// TwinCAT 3 PLC project PersistentData
// Title: ManagePersistentData
// Company: beckhoff.co.jp
// Author: Beckhoff Automation K.K.
// ProjectVersion: 1.0.0.1
// ProgramVersion: 3.1.4024.0
// libraries:
//   Tc2_IoFunctions, * (Beckhoff Automation GmbH)
//   Tc2_Standard, * (Beckhoff Automation GmbH)
//   Tc2_SUPS, * (Beckhoff Automation GmbH)
//   Tc2_System, * (Beckhoff Automation GmbH)
//   Tc2_Utilities, * (Beckhoff Automation GmbH)
//   Tc3_Module, * (Beckhoff Automation GmbH)
// project tree:
//   DUTs/ E_ShutdownMode.TcDUT, E_UPSState.TcDUT
//   / PlcTask.TcTTO
//   POUs/ FB_GenericUPS.TcPOU, FB_ShutDown.TcPOU, FB_SUPS_CX51x0.TcPOU, FB_UPS_STUB.TcPOU, iUPS.TcIO, MAIN.TcPOU
//   Project Information/ F_GetCompany.TcPOU, F_GetTitle.TcPOU, F_GetVersion.TcPOU
//   Version/ Global_Version.TcGVL
// real-time tasks:
//   TASK PlcTask: cycle T#10ms, priority 20, ADS port 350

CONFIGURATION PersistentData
    RESOURCE PLC ON TwinCAT3
        TASK PlcTask(INTERVAL := T#10ms, PRIORITY := 20);
        PROGRAM MAIN WITH PlcTask : MAIN;
    END_RESOURCE
END_CONFIGURATION

// ---- DUTs/E_ShutdownMode.TcDUT
{attribute 'qualified_only'}
{attribute 'strict'}
TYPE E_ShutdownMode :
(
	init := 0,			// system is working
	persistent_data,	// persist data
	shutting_down		// system shutting down
);
END_TYPE

// ---- DUTs/E_UPSState.TcDUT
{attribute 'qualified_only'}
{attribute 'strict'}
TYPE E_UPSState :
(
	init := 0,		// UPS not working
	on_power,		// power supplied normally
	on_battery,		// continue working on battery
	critical_error,	// system shutdown
	facility_error	// UPC failure
);
END_TYPE

// ---- Version/Global_Version.TcGVL
{attribute 'TcGenerated'}
{attribute 'no-analysis'}
{attribute 'linkalways'}
// This function has been automatically generated from the project information.
VAR_GLOBAL CONSTANT
	{attribute 'const_non_replaced'}
	stLibVersion_ManagePersistentData : ST_LibVersion := (iMajor := 1, iMinor := 0, iBuild := 0, iRevision := 1, nFlags := 0, sVersion := '1.0.0.1');
END_VAR

// ---- POUs/iUPS.TcIO
INTERFACE iUPS

(*
Method of saving persistent data
=================================================

Author
	: Takashi Ichihashi

Date
	: 02 Aug, 2023

Overview
===============

This method is assumed that persistent values are saved when ups running without online power.
"WritePersistentData" FB has to be executed explicily in case of GenericUPS is used. You might define this FB instance on this method.
If you use "SUPS", it might be saved persistent data automatically when power failed, so nothing need to be defined on this method.

*)
METHOD persist_data : BOOL
VAR_INPUT
END_VAR
END_METHOD

METHOD shutdown : BOOL
VAR_INPUT
END_VAR
END_METHOD

PROPERTY shutdown_delay : TIME
GET
END_GET
SET
END_SET
END_PROPERTY

PROPERTY UPSState : E_UPSState
GET
END_GET
END_PROPERTY

METHOD watch_status : BOOL
VAR_INPUT
END_VAR
END_METHOD

END_INTERFACE

// ---- POUs/MAIN.TcPOU
PROGRAM MAIN
VAR
	fbShutdown	:FB_ShutDown; // Safely shutdown feature
	fbUPS		:FB_SUPS_CX51x0; // UPS type for test use
END_VAR

fbUPS.shutdown_delay := T#3S;
fbShutdown(fbUPS := fbUPS);

END_PROGRAM

// ---- POUs/FB_ShutDown.TcPOU
FUNCTION_BLOCK FB_ShutDown
VAR_INPUT
	fbUPS			:iUPS;				// UPS interface	
END_VAR
VAR_OUTPUT
END_VAR
VAR
	eShutdownMode	:E_ShutdownMode;	// State machine when shutting down
END_VAR

// watch power fail
fbUPS.watch_status();

CASE fbUPS.UPSState OF 
	E_UPSState.on_battery:
		eShutdownMode := E_ShutdownMode.persistent_data;
	E_UPSState.critical_error:
		eShutdownMode := E_ShutdownMode.shutting_down;
	ELSE
		eShutdownMode := E_ShutdownMode.init;
END_CASE

CASE eShutdownMode OF 
	E_ShutdownMode.persistent_data:
		fbUPS.persist_data();
		IF fbUPS.UPSState = E_UPSState.facility_error THEN
			eShutdownMode := E_ShutdownMode.shutting_down;
		END_IF
	E_ShutdownMode.shutting_down:
		fbUPS.shutdown();
END_CASE

END_FUNCTION_BLOCK

// ---- POUs/FB_SUPS_CX51x0.TcPOU
FUNCTION_BLOCK FB_SUPS_CX51x0 IMPLEMENTS iUPS
VAR_INPUT
END_VAR
VAR_OUTPUT
END_VAR
VAR
	eUPSState 		:E_UPSState;
	tShutdownDelay	: TIME := T#1S;
	fbShutdownTimer	:Tc2_Standard.TON;
	fbS_UPS_CX51x0	:Tc2_SUPS.FB_S_UPS_CX51x0;
	fbShutdown		:FB_NT_QuickShutdown;
END_VAR

(*
Method of saving persistent data
=================================================

Author
	: Takashi Ichihashi

Date
	: 02 Aug, 2023

Overview
===============

This method is assumed that persistent values are saved when ups running without online power.
"WritePersistentData" FB has to be executed explicily in case of GenericUPS is used. You might define this FB instance on this method.
If you use "SUPS", it might be saved persistent data automatically when power failed, so nothing need to be defined on this method.

*)
METHOD persist_data : BOOL

IF fbS_UPS_CX51x0.eState = Tc2_SUPS.E_S_UPS_State.eSUPS_WaitForRecover THEN
	fbShutdownTimer(IN:=fbS_UPS_CX51x0.bPowerFailDetect, PT:=tShutdownDelay);
END_IF
END_METHOD

METHOD shutdown : BOOL
fbShutdown(START := TRUE);
END_METHOD

{warning 'add property implementation'}
PROPERTY shutdown_delay : TIME
GET
shutdown_delay := tShutdownDelay;
END_GET
SET
tShutdownDelay := shutdown_delay;
END_SET
END_PROPERTY

PROPERTY UPSState : E_UPSState
GET
UPSState := eUPSState;
END_GET
END_PROPERTY

METHOD watch_status : BOOL

fbS_UPS_CX51x0(eUpsMode := Tc2_SUPS.E_S_UPS_Mode.eSUPS_WrPersistData_NoShutdown);

CASE fbS_UPS_CX51x0.eState OF
	Tc2_SUPS.E_S_UPS_State.eSUPS_PowerOK:
		eUPSState := E_UPSState.on_power;
	Tc2_SUPS.E_S_UPS_State.eSUPS_PowerFailure:
		eUPSState := E_UPSState.on_battery;
	Tc2_SUPS.E_S_UPS_State.eSUPS_WritePersistentData:
		eUPSState := E_UPSState.on_battery;
	Tc2_SUPS.E_S_UPS_State.eSUPS_WaitForRecover:
		IF fbShutdownTimer.Q THEN
			eUPSState := E_UPSState.critical_error;
		ELSE
			eUPSState := E_UPSState.on_battery;
		END_IF
	Tc2_SUPS.E_S_UPS_State.eSUPS_WaitForPowerOFF:
		eUPSState := E_UPSState.critical_error;
	Tc2_SUPS.E_S_UPS_State.eSUPS_QuickShutdown:
		eUPSState := E_UPSState.critical_error;
	ELSE
		eUPSState := E_UPSState.init;
END_CASE
END_METHOD

END_FUNCTION_BLOCK

// ---- POUs/FB_GenericUPS.TcPOU
FUNCTION_BLOCK FB_GenericUPS IMPLEMENTS iUPS
VAR_INPUT
END_VAR
VAR_OUTPUT
END_VAR
VAR
END_VAR

{warning 'add method implementation '}
METHOD persist_data : BOOL
END_METHOD

{warning 'add method implementation '}
METHOD shutdown : BOOL
END_METHOD

{warning 'add property implementation'}
PROPERTY UPSState : E_UPSState
GET
END_GET
SET
END_SET
END_PROPERTY

{warning 'add method implementation '}
METHOD watch_status : BOOL
END_METHOD

END_FUNCTION_BLOCK

// ---- POUs/FB_UPS_STUB.TcPOU
FUNCTION_BLOCK FB_UPS_STUB IMPLEMENTS iUPS
VAR_INPUT
END_VAR
VAR_OUTPUT
END_VAR
VAR
	eUPSState :E_UPSState;
	tShutdownDelay	: TIME := T#5S;
	test_timer :Tc2_Standard.TON;
END_VAR

{warning 'add method implementation '}
METHOD persist_data : BOOL
END_METHOD

{warning 'add method implementation '}
METHOD shutdown : BOOL
END_METHOD

{warning 'add property implementation'}
PROPERTY shutdown_delay : TIME
GET
shutdown_delay := tShutdownDelay;
END_GET
SET
tShutdownDelay := shutdown_delay;
END_SET
END_PROPERTY

{warning 'add property implementation'}
PROPERTY UPSState : E_UPSState
GET
UPSState := eUPSState;
END_GET
END_PROPERTY

{warning 'add method implementation '}
METHOD watch_status : BOOL
IF eUPSState = E_UPSState.on_battery THEN
	test_timer.PT := tShutdownDelay;
ELSE
	test_timer.PT := T#15S;
END_IF

test_timer(IN := NOT test_timer.Q);

IF test_timer.Q THEN
	CASE eUPSState OF
		E_UPSState.init:
			eUPSState := E_UPSState.on_power;
		E_UPSState.on_power:
			eUPSState := E_UPSState.on_battery;
		E_UPSState.critical_error:
			eUPSState := E_UPSState.init;
	END_CASE
END_IF
END_METHOD

END_FUNCTION_BLOCK

// ---- Project Information/F_GetCompany.TcPOU
// This function has been automatically generated from the project information.
{attribute 'signature_flag' := '1073741824'}
{attribute 'TcGenerated'}
{attribute 'no-analysis'}
FUNCTION F_GetCompany : WSTRING
VAR_INPUT
	
END_VAR

F_GetCompany := "beckhoff.co.jp";

END_FUNCTION

// ---- Project Information/F_GetTitle.TcPOU
// This function has been automatically generated from the project information.
{attribute 'signature_flag' := '1073741824'}
{attribute 'TcGenerated'}
{attribute 'no-analysis'}
FUNCTION F_GetTitle : WSTRING
VAR_INPUT
	
END_VAR

F_GetTitle := "ManagePersistentData";

END_FUNCTION

// ---- Project Information/F_GetVersion.TcPOU
// This function has been automatically generated from the project information.
{attribute 'signature_flag' := '1073741824'}
{attribute 'TcGenerated'}
{attribute 'no-analysis'}
FUNCTION F_GetVersion : ST_LibVersion
VAR_INPUT
	
END_VAR

F_GetVersion.iMajor := 1;
F_GetVersion.iMinor := 0;
F_GetVersion.iBuild := 0;
F_GetVersion.iRevision := 1;
F_GetVersion.sVersion := '1.0.0.1';
F_GetVersion.nFlags := 0;

END_FUNCTION
